screen "Storage" 1280x740, template "Template_1"
   on GenerateScreen: SetTag("Tag_ScreenNumber", 3)
   Button "Back" at 1,1 size 159x47; TextOff 'Back'
      on Release: ActivateScreen("Root screen", 0)
   Button "Button_1" at 905,545 size 96x58; TextOff '1'
      on Activate: SetTag("user target position", 0); SetBit("deploy")
      Appearance <- "[0]"
   Button "Button_2" at 798,545 size 96x58; TextOff '2'
      on Activate: SetTag("user target position", 1); SetBit("deploy")
      Appearance <- "[1]"
   Button "Button_3" at 692,545 size 96x58; TextOff '3'
      on Activate: SetTag("user target position", 2); SetBit("deploy")
      Appearance <- "[2]"
   Button "Button_4" at 585,545 size 96x58; TextOff '4'
      on Activate: SetTag("user target position", 3); SetBit("deploy")
      Appearance <- "[3]"
   Button "Button_5" at 479,545 size 96x58; TextOff '5'
      on Activate: SetTag("user target position", 4); SetBit("deploy")
      Appearance <- "[4]"
   Button "Button_6" at 373,545 size 96x58; TextOff '6'
      on Activate: SetTag("user target position", 5); SetBit("deploy")
      Appearance <- "[5]"
   Button "Button_7" at 266,545 size 96x58; TextOff '7'
      on Activate: SetTag("user target position", 6); SetBit("deploy")
      Appearance <- "[6]"
   Button "Button_8" at 160,545 size 96x58; TextOff '8'
      on Activate: SetTag("user target position", 7); SetBit("deploy")
      Appearance <- "[7]"
   Button "Button_9" at 54,545 size 96x58; TextOff '9'
      on Activate: SetTag("user target position", 8); SetBit("deploy")
      Appearance <- "[8]"
   Button "Button_10" at 905,464 size 96x58; TextOff '10'
      on Activate: SetTag("user target position", 9); SetBit("deploy")
      Appearance <- "[9]"
   Button "Button_11" at 798,464 size 96x58; TextOff '11'
      on Activate: SetTag("user target position", 10); SetBit("deploy")
      Appearance <- "[10]"
   Button "Button_12" at 692,464 size 96x58; TextOff '12'
      on Activate: SetTag("user target position", 11); SetBit("deploy")
      Appearance <- "[11]"
   Button "Button_13" at 585,464 size 96x58; TextOff '13'
      on Activate: SetTag("user target position", 12); SetBit("deploy")
      Appearance <- "[12]"
   Button "Button_14" at 479,464 size 96x58; TextOff '14'
      on Activate: SetTag("user target position", 13); SetBit("deploy")
      Appearance <- "[13]"
   Button "Button_15" at 373,464 size 96x58; TextOff '15'
      on Activate: SetTag("user target position", 14); SetBit("deploy")
      Appearance <- "[14]"
   Button "Button_16" at 266,464 size 96x58; TextOff '16'
      on Activate: SetTag("user target position", 15); SetBit("deploy")
      Appearance <- "[15]"
   Button "Button_17" at 160,464 size 96x58; TextOff '17'
      on Activate: SetTag("user target position", 16); SetBit("deploy")
      Appearance <- "[16]"
   Button "Button_18" at 54,464 size 96x58; TextOff '18'
      on Activate: SetTag("user target position", 17); SetBit("deploy")
      Appearance <- "[17]"
   Button "Button_19" at 905,384 size 96x58; TextOff '19'
      on Activate: SetTag("user target position", 18); SetBit("deploy")
      Appearance <- "[18]"
   Button "Button_20" at 798,384 size 96x58; TextOff '20'
      on Activate: SetTag("user target position", 19); SetBit("deploy")
      Appearance <- "[19]"
   Button "Button_21" at 692,384 size 96x58; TextOff '21'
      on Activate: SetTag("user target position", 20); SetBit("deploy")
      Appearance <- "[20]"
   Button "Button_22" at 585,384 size 96x58; TextOff '22'
      on Activate: SetTag("user target position", 21); SetBit("deploy")
      Appearance <- "[21]"
   Button "Button_23" at 479,384 size 96x58; TextOff '23'
      on Activate: SetTag("user target position", 22); SetBit("deploy")
      Appearance <- "[22]"
   Button "Button_24" at 373,384 size 96x58; TextOff '24'
      on Activate: SetTag("user target position", 23); SetBit("deploy")
      Appearance <- "[23]"
   Button "Button_25" at 266,384 size 96x58; TextOff '25'
      on Activate: SetTag("user target position", 24); SetBit("deploy")
      Appearance <- "[24]"
   Button "Button_26" at 160,384 size 96x58; TextOff '26'
      on Activate: SetTag("user target position", 25); SetBit("deploy")
      Appearance <- "[25]"
   Button "Button_27" at 54,384 size 96x58; TextOff '27'
      on Activate: SetTag("user target position", 26); SetBit("deploy")
      Appearance <- "[26]"
   Button "Button_28" at 905,304 size 96x58; TextOff '28'
      on Activate: SetTag("user target position", 27); SetBit("deploy")
      Appearance <- "[27]"
   Button "Button_29" at 798,304 size 96x58; TextOff '29'
      on Activate: SetTag("user target position", 28); SetBit("deploy")
      Appearance <- "[28]"
   Button "Button_30" at 692,304 size 96x58; TextOff '30'
      on Activate: SetTag("user target position", 29); SetBit("deploy")
      Appearance <- "[29]"
   Button "Button_31" at 585,304 size 96x58; TextOff '31'
      on Activate: SetTag("user target position", 30); SetBit("deploy")
      Appearance <- "[30]"
   Button "Button_32" at 479,304 size 96x58; TextOff '32'
      on Activate: SetTag("user target position", 31); SetBit("deploy")
      Appearance <- "[31]"
   Button "Button_33" at 373,304 size 96x58; TextOff '33'
      on Activate: SetTag("user target position", 32); SetBit("deploy")
      Appearance <- "[32]"
   Button "Button_34" at 266,304 size 96x58; TextOff '34'
      on Activate: SetTag("user target position", 33); SetBit("deploy")
      Appearance <- "[33]"
   Button "Button_35" at 160,304 size 96x58; TextOff '35'
      on Activate: SetTag("user target position", 34); SetBit("deploy")
      Appearance <- "[34]"
   Button "Button_36" at 54,304 size 96x58; TextOff '36'
      on Activate: SetTag("user target position", 35); SetBit("deploy")
      Appearance <- "[35]"
   Button "Button_37" at 905,223 size 96x58; TextOff '37'
      on Activate: SetTag("user target position", 36); SetBit("deploy")
      Appearance <- "[36]"
   Button "Button_38" at 798,223 size 96x58; TextOff '38'
      on Activate: SetTag("user target position", 37); SetBit("deploy")
      Appearance <- "[37]"
   Button "Button_39" at 692,223 size 96x58; TextOff '39'
      on Activate: SetTag("user target position", 38); SetBit("deploy")
      Appearance <- "[38]"
   Button "Button_40" at 585,223 size 96x58; TextOff '40'
      on Activate: SetTag("user target position", 39); SetBit("deploy")
      Appearance <- "[39]"
   Button "Button_41" at 479,223 size 96x58; TextOff '41'
      on Activate: SetTag("user target position", 40); SetBit("deploy")
      Appearance <- "[40]"
   Button "Button_42" at 373,223 size 96x58; TextOff '42'
      on Activate: SetTag("user target position", 41); SetBit("deploy")
      Appearance <- "[41]"
   Button "Button_43" at 266,223 size 96x58; TextOff '43'
      on Activate: SetTag("user target position", 42); SetBit("deploy")
      Appearance <- "[42]"
   Button "Button_44" at 160,223 size 96x58; TextOff '44'
      on Activate: SetTag("user target position", 43); SetBit("deploy")
      Appearance <- "[43]"
   Button "Button_45" at 54,223 size 96x58; TextOff '45'
      on Activate: SetTag("user target position", 44); SetBit("deploy")
      Appearance <- "[44]"
   Button "Button_46" at 905,145 size 96x58; TextOff '46'
      on Activate: SetTag("user target position", 45); SetBit("deploy")
      Appearance <- "[45]"
   Button "Button_47" at 798,145 size 96x58; TextOff '47'
      on Activate: SetTag("user target position", 46); SetBit("deploy")
      Appearance <- "[46]"
   Button "Button_48" at 692,145 size 96x58; TextOff '48'
      on Activate: SetTag("user target position", 47); SetBit("deploy")
      Appearance <- "[47]"
   Button "Button_49" at 585,145 size 96x58; TextOff '49'
      on Activate: SetTag("user target position", 48); SetBit("deploy")
      Appearance <- "[48]"
   Button "Button_50" at 479,145 size 96x58; TextOff '50'
      on Activate: SetTag("user target position", 49); SetBit("deploy")
      Appearance <- "[49]"
   Button "Button_51" at 373,145 size 96x58; TextOff '51'
      on Activate: SetTag("user target position", 50); SetBit("deploy")
      Appearance <- "[50]"
   Button "Button_52" at 266,145 size 96x58; TextOff '52'
      on Activate: SetTag("user target position", 51); SetBit("deploy")
      Appearance <- "[51]"
   Button "Button_53" at 160,145 size 96x58; TextOff '53'
      on Activate: SetTag("user target position", 52); SetBit("deploy")
      Appearance <- "[52]"
   Button "Button_54" at 54,145 size 96x58; TextOff '54'
      on Activate: SetTag("user target position", 53); SetBit("deploy")
      Appearance <- "[53]"
   IOField "I/O field_1" at 1212,223 size 40x32; FormatPattern 99
      ProcessValue <- "cap"
   TextField "Text field_1" at 1029,226 size 177x25; Text 'Storage capacity :'
   Switch "Switch_1" at 1061,528 size 151x74; CaptionText 'Load'; TextOff 'to Exit'; TextOn 'to Storage'
      ProcessValue <- "Load to storage"
   TextField "Text field_2" at 1029,286 size 177x25; Text 'Blue pack stored :'
   IOField "I/O field_2" at 1212,285 size 40x32; FormatPattern 99
      ProcessValue <- "blue item stored"
   TextField "Text field_3" at 1029,346 size 189x25; Text 'green pack stored :'
   IOField "I/O field_3" at 1212,346 size 40x32; FormatPattern 99
      ProcessValue <- "green item stored"
   TextField "Text field_4" at 1032,407 size 140x25; Text 'Crane Uptime:'
   IOField "I/O field_4" at 1212,400 size 40x32; FormatPattern 99999
      ProcessValue <- "crane uptime"

screen "packing" 1280x740, template "Template_1"
   on GenerateScreen: SetTag("Tag_ScreenNumber", 4)
   Button "Back" at 1,1 size 159x47; TextOff 'Back'
      on Release: ActivateScreen("Root screen", 0)
   Rectangle "Rectangle_2" at 136,124 size 96x488
      Appearance <- "Packaging Blue Exit Convoyer 1"
   Rectangle "Rectangle_1" at 248,307 size 96x305
      Appearance <- "Packaging Blue Convoyer"
   Circle "Circle_1" at 336,350 size 28x28
      Appearance <- "Packaging Blue(Clamp)"
   Circle "Circle_2" at 118,350 size 28x28
      Appearance <- "Packaging Blue Palet Sensor"
   TextField "Text field_1" at 8,351 size 121x22; Text 'Palet at place'
   TextField "Text field_2" at 348,386 size 56x22; Text 'Clamp'
   Rectangle "Rectangle_3" at 524,124 size 96x488
      Appearance <- "Packaging Green Exit Convoyer"
   Rectangle "Rectangle_4" at 636,307 size 96x305
      Appearance <- "Packaging Green Convoyer"
   Circle "Circle_3" at 724,350 size 28x28
      Appearance <- "Packaging Green (Clamp)"
   Circle "Circle_4" at 506,350 size 28x28
      Appearance <- "Packaging Blue Palet Sensor"
   TextField "Text field_3" at 398,350 size 121x22; Text 'Palet at place'
   TextField "Text field_4" at 736,386 size 56x22; Text 'Clamp'
   Button "Button_1" at 574,571 size 115x42; TextOff 'Reset'
      on Activate: ResetBit("entry convoyer packing green ready"); ResetBit("exit convoyer packing green ready"); ResetBit("ready to pack 2"); ResetBit("reset packer 2")
      on Press: SetBit("reset packer 2")
   IOField "I/O field_1" at 115,304 size 31x32; FormatPattern 9
      ProcessValue <- "Item in blue pack"
   IOField "I/O field_2" at 505,304 size 31x32; FormatPattern 9
      ProcessValue <- "Item in green pack"
   TextField "Text field_5" at 203,629 size 88x25; Text 'Blue line'
   TextField "Text field_6" at 585,626 size 102x25; Text 'Green line'
   TextField "Text field_7" at 839,120 size 217x25; Text 'green pack produced :'
   TextField "Text field_8" at 839,190 size 204x25; Text 'blue pack produced :'
   TextField "Text field_9" at 839,331 size 206x25; Text 'blue packer up time :'
   TextField "Text field_10" at 839,260 size 219x25; Text 'green packer up time :'
   IOField "I/O field_3" at 1044,118 size 96x32; FormatPattern 99999
      ProcessValue <- "green pack produced"
   IOField "I/O field_4" at 1044,188 size 96x32; FormatPattern 99999
      ProcessValue <- "Blue pack produced"
   IOField "I/O field_5" at 1044,258 size 96x32; FormatPattern 99999
      ProcessValue <- "counter packing 1 uptime"
   IOField "I/O field_6" at 1044,329 size 96x32; FormatPattern 99999
      ProcessValue <- "uptime blue packing"
   Button "Button_2" at 181,571 size 115x42; TextOff 'Reset'
      on Activate: ResetBit("entry convoyer packing blue ready"); ResetBit("exit convoyer packing blue ready"); ResetBit("reset packer 1")
      on Press: SetBit("reset packer 1")

screen "System screens" 1280x740, template "Template_1"
   on GenerateScreen: SetTag("Tag_ScreenNumber", 6)
   Button "Back" at 1,1 size 159x47; TextOff 'Back'
      on Release: ActivateScreen("Root screen", 0)
   Button "HmiScreenItemData" at 36,95 size 159x47; TextOff 'System settings'; PictureOff "Navigates to System settings for TP1200 Comfort 17.0.0.0"; PictureOn "Navigates to System settings for TP1200 Comfort 17.0.0.0"
      on Release: ActivateScreen("System settings", 0)

screen "System settings" 1280x740, template "Template_1"
   on GenerateScreen: SetTag("Tag_ScreenNumber", 7)
   Button "Calibrate screen" at 36,95 size 159x47; TextOff 'Calibrate screen'
      on Release: function_bc3e350c()
   Button "Clean screen" at 36,154 size 159x47; TextOff 'Clean screen'
      on Release: function_be740847(30)
   Button "Back" at 1,1 size 159x47; TextOff 'Back'
      on Release: ActivateScreen("System screens", 0)
*)